TYPE DINT_LENGTH : DINT(0..2147483647); END_TYPE

(* stored: Version 1.1.0.1
   DUT DINT_LENGTH: Id {370b5060-1d88-4d8d-aceb-c3b1f396a9a6} *)
